TYPE OutStream :
STRUCT
	ForceFan1_SetSpeed: REAL;
	ForceFan2_SetSpeed: REAL;
	ForceFan3_SetSpeed: REAL;
	CondensePump_SetSpeed: REAL;
	SupplyPump_SetSpeed: REAL;
	CircularPump_OutFlow: REAL;
	LPHeaterValve_SetPercent: REAL;
	AirEjectorValve_SetPercent: REAL;
	HPHeaterValve_SetPercent: REAL;
	TurbineValve_SetPercent: REAL;
END_STRUCT
END_TYPE

(* stored: Version 1.1.0.1, ProductVersion 3.1.4024.4
   DUT OutStream: Id {756ac912-a9ec-4daa-b1e4-0f27d2726c76} *)
